// TIA Portal V15 export
// export: Created 2018-02-11T06:46:14.3598303Z, ExportSetting None, DisplayName Totally Integrated Automation Portal, DisplayVersion V15, DisplayName TIA Portal Openness, DisplayVersion V15, DisplayName TIA Portal Teamcenter Gateway, DisplayVersion V15, DisplayName SINAMICS Startdrive Advanced, DisplayVersion V15, DisplayName G110M, G120, G120C, G120D, G120P, DisplayVersion V15, DisplayName G130, G150, S120, S150, SINAMICS MV, DisplayVersion V15, DisplayName STEP 7 Professional, DisplayVersion V15, DisplayName WinCC Professional, DisplayVersion V15, DisplayName SIMATIC Visualization Architect, DisplayVersion V15
FUNCTION "Workshop2_FC" : Void   // FC2, LAD
{ S7_Optimized_Access := 'TRUE' }
// stored: SetENOAutomatically False
   VAR_INPUT
      WaterLevel : Int;
      OilLevel : Int;
   END_VAR
BEGIN

REGION Network 1
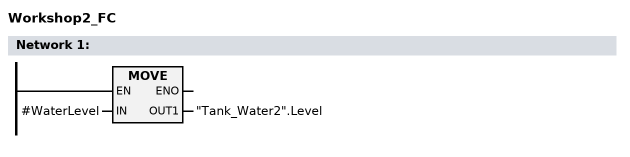
   RUNG wire#powerrail
      Move(in := #WaterLevel, out1 => "Tank_Water2".Level)
   END_RUNG
   // the same network as SCL:
   "Tank_Water2".Level := #WaterLevel;
END_REGION
END_FUNCTION
